{attribute 'qualified_only'}
{attribute 'strict'}
{attribute 'to_string'}
TYPE E_MotorStatus :
(
	Uit := 0,
	Aan := 1,
	Error:= 2
);
END_TYPE

(* stored: Version 1.1.0.1
   DUT E_MotorStatus: Id {405a818c-d009-4827-9789-ca6436a46b39} *)
